FUNCTION RawToCurrent : REAL
VAR_INPUT
	raw : UINT;            // 0 to 5000
END_VAR


RawToCurrent := UINT_TO_REAL(raw) * 0.001;  // → 0.00 to 5.00 A

END_FUNCTION

(* stored: Version 1.1.0.1
   POU RawToCurrent: Id {1b9b501d-b8f1-4179-abec-44f33dc96542}, SpecialFunc None *)
